Yaskawa INFORM job: R2-ST1-SAFE.JBI

/JOB
//NAME R2-ST1-SAFE
///FOLDERNAME FOLDER001
//POS
///NPOS 4,4,0,0,3,0
///TOOL 0
///POSTYPE PULSE
///PULSE
C00000=-3570,-156343,-136271,3723,37683,81363
C00001=-3570,-156343,-136271,3723,37683,81363
C00002=-3570,-156343,-136271,3723,37683,81363
C00003=-3570,-156343,-136271,3723,37683,81364
BC00000=85972,867731,452132
BC00001=85972,867731,452132
BC00002=85972,867731,452132
BC00003=85972,285995,452132
///POSTYPE BASE
///RECTAN
///RCONF 0,0,0,0,0,0,0,0,0,0,0,0,0,0,0,0,0,0,0,0,0,0,0,0
BP00001=1748.393,5381.174,256.888
///POSTYPE ROBOT
BP00002=0.000,-559.016,0.000
BP00003=0.000,-559.016,0.000
//INST
///DATE 2023/07/10 17:15
///ATTR SC,RW
///GROUP1 RB1,BS1
NOP
SFTOF
REFP 1 C00000 BC00000
GETS PX001 $PX011
CNVRT PX001 PX001 RF
GETS PX002 $PX001
CNVRT PX002 PX002 RF
SUB BP002 BP001
SET BP003 BP002
SFTON BP003
MOVJ C00001 BC00001 VJ=50.00
SFTOF
SETE BP003 (1) 0
SETE BP003 (3) 0
SFTON BP003
MOVJ C00002 BC00002 VJ=100.00
SFTOF
MOVJ C00003 BC00003 VJ=100.00
END
